{attribute 'qualified_only'}
VAR_GLOBAL
	
END_VAR

(* stored: Version 1.1.0.1, ProductVersion 3.1.4024.12
   GVL GVL_Interlock: Id {8a699700-4d69-4643-8506-8218cdab8ca3} *)
